PROGRAM MAIN
VAR
END_VAR

MainASR();

END_PROGRAM

(* stored: Version 1.1.0.1
   POU MAIN: Id {a71e5ec2-15ed-4b94-967c-544b000f6e0f}, SpecialFunc None *)
